FUNCTION_BLOCK overcurrentV2_IO_1_backup2 (* Composite Function Block Type *)
  (* Standard: 61499-2 *)
  (* Version 0.0, 23/05/2016, Chen-Wei, nxtControl GmbH, template *)
  PACKAGE Main;
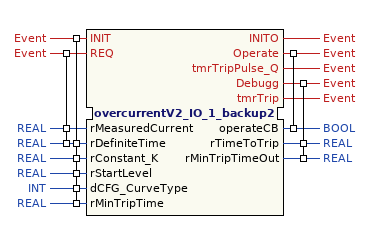
  EVENT_INPUT
    INIT WITH rDefiniteTime, rConstant_K, rStartLevel, dCFG_CurveType, rMinTripTime; (* Initialization Request *)
    REQ WITH rMeasuredCurrent, rDefiniteTime; (* Normal Execution Request *)
  END_EVENT
  EVENT_OUTPUT
    INITO; (* Initialization Confirm *)
    Operate WITH operateCB; (* Delayed Event *)
    tmrTripPulse_Q; (* Delayed Event *)
    Debugg WITH rTimeToTrip, rMinTripTimeOut;
    tmrTrip; (* Execution Confirmation *)
  END_EVENT
  VAR_INPUT
    rMeasuredCurrent : REAL; (* Input event qualifier *)
    rDefiniteTime : REAL;
    rConstant_K : REAL;
    rStartLevel : REAL;
    dCFG_CurveType : INT;
    rMinTripTime : REAL;
  END_VAR
  VAR_OUTPUT
    operateCB : BOOL; (* Output event qualifier *)
    rTimeToTrip : REAL;
    rMinTripTimeOut : REAL;
  END_VAR
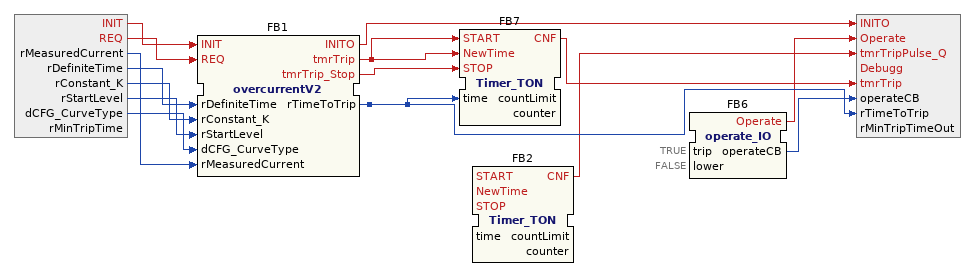
  FBS
    FB6 : operate_IO(trip := TRUE, lower := FALSE);
    FB1 : overcurrentV2;
    FB7 : Timer_TON;
    FB2 : Timer_TON;
  END_FBS
  EVENT_CONNECTIONS
    INIT TO FB1.INIT;
    FB6.Operate TO Operate;
    REQ TO FB1.REQ;
    FB2.CNF TO tmrTripPulse_Q;
    FB1.INITO TO INITO;
    FB1.tmrTrip TO FB7.NewTime;
    FB1.tmrTrip TO FB7.START;
    FB1.tmrTrip_Stop TO FB7.STOP;
    FB7.CNF TO tmrTrip;
  END_CONNECTIONS
  DATA_CONNECTIONS
    FB6.operateCB TO operateCB;
    rDefiniteTime TO FB1.rDefiniteTime;
    rConstant_K TO FB1.rConstant_K;
    rStartLevel TO FB1.rStartLevel;
    dCFG_CurveType TO FB1.dCFG_CurveType;
    rMeasuredCurrent TO FB1.rMeasuredCurrent;
    FB1.rTimeToTrip TO rTimeToTrip;
    FB1.rTimeToTrip TO FB7.time;
  END_CONNECTIONS
END_FUNCTION_BLOCK
